(* IEC 61131-3 sources: STLLVM-Examples/, 8 files *)

(* ---- binary_search.st ---- *)
PROGRAM binary_search
  VAR_INPUT x : INT; END_VAR
  VAR_INPUT arr : ARRAY[0..9] OF INT; END_VAR
  VAR_OUTPUT idx : INT; END_VAR
  VAR_TEMP
    i : INT;
    first : INT := 0;
    last : INT := 9;
    mid : INT;
  END_VAR

FOR i := 0 TO 8 DO
  __ASSUME arr[i] <= arr[i + 1];
END_FOR

idx := -1;
WHILE first <= last DO
  mid := (first + last) / 2;
  IF arr[mid] = x THEN
    idx := mid;
    EXIT;
  ELSIF arr[mid] > x THEN
    last := mid - 1;
  ELSE
    first := mid + 1;
  END_IF
END_WHILE

IF idx <> -1 THEN
  IF arr[idx] <> x THEN
    __UNREACHABLE;
  END_IF
END_IF

END_PROGRAM

(* ---- boiler.st ---- *)
PROGRAM boiler
VAR_INPUT
  temperature : INT;
END_VAR
VAR_OUTPUT
  heater_on : BOOL;
END_VAR
VAR
  last_temperature : INT;
END_VAR
VAR_TEMP CONSTANT
  target_temperature : INT := 100;
  hysteresis : INT := 5;
END_VAR

IF temperature > last_temperature THEN
  // Rising temperature.
  IF temperature > target_temperature + hysteresis THEN
    heater_on := FALSE;
  ELSE
    heater_on := TRUE;
  END_IF
ELSE
  // Falling temperature.
  IF temperature < target_temperature THEN
    heater_on := TRUE;
  ELSE
    heater_on := FALSE;
  END_IF
END_IF

last_temperature := temperature;
IF temperature > target_temperature + hysteresis AND heater_on THEN
__UNREACHABLE;
END_IF

END_PROGRAM

(* ---- buffer.st ---- *)
PROGRAM buffer
  VAR_INPUT value : INT; END_VAR
  VAR_INPUT offset : INT; END_VAR
  VAR_GLOBAL buf : ARRAY [0..1024] OF INT; END_VAR
  VAR cur_pos : INT := 0; END_VAR

IF offset < 0 THEN RETURN; END_IF
IF cur_pos + offset > 1024 THEN RETURN; END_IF;

cur_pos := cur_pos + offset;
buf[cur_pos] := value;

END_PROGRAM

(* ---- copy-loop-bug.st ---- *)
PROGRAM pcopy
VAR_INPUT i : INT; END_VAR
VAR_OUTPUT o : INT; END_VAR

o := 0;
WHILE i > 0 DO
  i := i - 1;
  o := o + 1;
END_WHILE

END_PROGRAM

(* ---- copy-loop-fixed.st ---- *)
PROGRAM pcopy
VAR_INPUT i : INT; END_VAR
VAR_OUTPUT o : INT; END_VAR

o := 0;
IF i > 0 THEN
  WHILE i > 0 DO
    i := i - 1;
    o := o + 1;
  END_WHILE
ELSE
  WHILE i < 0 DO
    i := i + 1;
    o := o - 1;
  END_WHILE
END_IF

END_PROGRAM

(* ---- copy.st ---- *)
PROGRAM pcopy
VAR_INPUT i : INT; END_VAR
VAR_OUTPUT o : INT; END_VAR

o := i;

END_PROGRAM

(* ---- deref.st ---- *)
TYPE
  IntRef : REF_TO INT;
END_TYPE

PROGRAM deref
  VAR_INPUT ptr : IntRef; END_VAR
  VAR_OUTPUT out : INT; END_VAR

  out := ptr^;
END_PROGRAM

(* ---- smooth.st ---- *)
PROGRAM smooth
  VAR_INPUT in_data : ARRAY[1..10] OF INT; END_VAR
  VAR_OUTPUT out_data : ARRAY[1..10] OF INT; END_VAR
  VAR_TEMP i, j : INT; val : INT; END_VAR

FOR i := 1 TO 10 DO
  val := 0;
  FOR j := i - 1 TO i + 1 DO
    IF j >= 1 AND j <= 10 THEN
      val := val + in_data[i] / ABS(i - j);
    END_IF;
  END_FOR
  out_data[i] := val / 2;
END_FOR

END_PROGRAM
